METHOD M_AlarmManagement
//////////////////
// Manages Sepam Alarms. Alarms opens HT CB until Sepam manual Reset. Warning Opens CB-L but does not maintain warning.
/////////////////

VAR 
	// Method local variables (reinitialized at each cycle) 
	FB_AlarmCodeManager 	: FB_AlarmCodeManager; 
 	ComWarning				: BOOL;
	ComAlarms				: BOOL;
END_VAR
// ALARM CODE //
	FB_AlarmCodeManager(
		bAlarm1			:= MesDataExd.MesData.MesAlarmCom,			// Com alarm
		bAlarm2			:= MesDataExd.MesData.MesFault_Major,				// True := Major fault : cannot recover
		bAlarm3			:= MesDataExd.MesData.MesAlarm_AcOff,				// True := AC off		
		bAlarm4			:= MesDataExd.MesData.MesAlarm_GeneralOff,			// True := Imminent shut down
		bAlarm5			:= MesDataExd.MesData.MesFault_Bat,					// True := Battery disconnected
		bAlarm6			:= MesDataExd.MesData.MesFault_Charger,				// True := Charger out of order										 
		bAlarm7			:= MesDataExd.MesData.MesFault_12V,					// True := 12V absent 
		bAlarm8			:= MesDataExd.MesData.MesFault_48V,					// True := 48V absent
		bAlarm9			:= MesDataExd.MesData.MesToggleRead,				// True := AC power supply low 
		bAlarm10		:= FALSE, 									//										
		bAlarm11		:= FALSE,                                   //
		bAlarm12		:= FALSE,                                   //
		bAlarm13		:= FALSE,                                   //
		bAlarm14		:= FALSE,                                   //
		bAlarm15		:= FALSE, 									// 
		wAlarmCode		=>MesDataExd.MesData.MesAlarmCode);		

// WARNING CODE //
	FB_AlarmCodeManager(
		bAlarm1			:= MesDataExd.MesData.MesFault_Minor,				// True := Minor fault (overtemp, overcurrent, overvolt)
		bAlarm2			:= MesDataExd.MesData.MesAlarm_Ulow ,		// Battery  Capacity is low 
		bAlarm4			:= FALSE,									//
		bAlarm5			:= FALSE,									//
		bAlarm6			:= FALSE,									//
		bAlarm7			:= FALSE,									// 
		bAlarm8			:= FALSE,									// 
		bAlarm9			:= FALSE,									// 
		bAlarm10		:= FALSE,									// 
		bAlarm11		:= FALSE,									// 
		bAlarm12		:= FALSE,									// 
		bAlarm13		:= FALSE,									// 
		bAlarm14		:= FALSE,									// 
		bAlarm15		:= FALSE,									// 
		wAlarmCode		=>MesDataExd.MesData.MesWarningCode);					

// EVENT CODE //
	FB_AlarmCodeManager(
		bAlarm1			:=FALSE, 									// 
		bAlarm2			:=FALSE, 									// 
		bAlarm3			:=FALSE, 									// 
		bAlarm4			:=FALSE, 									// 
		bAlarm5			:=FALSE, 									//
		bAlarm6			:=FALSE,        							//
		bAlarm7			:=FALSE,        							//
		bAlarm8			:=FALSE,        							//
		bAlarm9			:=FALSE,        							//
		bAlarm10		:=FALSE, 									//
		bAlarm11		:=FALSE,        							//
		bAlarm12		:=FALSE,        							//
		bAlarm13		:=FALSE,        							//
		bAlarm14		:=FALSE,        							//
		bAlarm15		:=FALSE, 									//
		wAlarmCode		=> MesDataExd.MesData.MesEventCode);
END_METHOD

METHOD M_Evaluate
VAR_INPUT
END_VAR

VAR
END_VAR
END_METHOD

METHOD M_Read
//////////////////
//  Method Calls 
/////////////////

VAR_INPUT
	
END_VAR
VAR 
	MW					: FB_MergeWordsToFloat;
	MW_1				: FB_MergeWordsToDint;
END_VAR
// CP-Read / Write 


IF MesDataExd.MesData.MesCP_Read  THEN		
	
	FB_ModbusRead[1]
		(
			nTCPPort		:= ParamTcpPort,
			ClockRead		:= MesDataExd.MesData.MesCP_Read AND ClockRead, 
			Reset			:= CmdClearFault_G OR IN_CmdReset_L,
			sIPAddr			:= ParamIPAddress ,
			nUnitID			:= 1, 
			tTimeout		:= T#5S,
			nQuantity		:= 1, 
			nMBAddr			:= 44000 , 
			cbLength		:= SIZEOF(MesBlock1_Temp) , 
			pDestAddr		:= ADR(MesBlock1_Temp) , 
			ModbusReadAlarm	=> AX_ModbusReadAlarm[1] , 
			ErrorId			=> AX_ModbusReadAlarmId[1]
		);
		
	FB_ModbusRead[2]
		(
			nTCPPort		:= ParamTcpPort,
			ClockRead		:= MesDataExd.MesData.MesCP_Read AND ClockRead, 
			Reset			:= CmdClearFault_G OR IN_CmdReset_L,
			sIPAddr			:= ParamIPAddress ,
			nUnitID			:= 1, 
			tTimeout		:= T#5S,
			nQuantity		:= 9, 
			nMBAddr			:= 44100 , 
			cbLength		:= SIZEOF(MesBlock2_Temp) , 
			pDestAddr		:= ADR(MesBlock2_Temp) , 
			ModbusReadAlarm	=> AX_ModbusReadAlarm[2], 
			ErrorId			=> AX_ModbusReadAlarmId[2]
		);
		
	FB_ModbusRead[3]
		(
			nTCPPort		:= ParamTcpPort,
			ClockRead		:= MesDataExd.MesData.MesCP_Read AND ClockRead	, 
			Reset			:= CmdClearFault_G OR IN_CmdReset_L,
			sIPAddr			:= ParamIPAddress ,
			nUnitID			:= 1, 
			tTimeout		:= T#5S,
			nQuantity		:= 6, 
			nMBAddr			:= 44150 , 
			cbLength		:= SIZEOF(MesBlock3_Temp) , 
			pDestAddr		:= ADR(MesBlock3_Temp) , 
			ModbusReadAlarm	=> AX_ModbusReadAlarm[3], 
			ErrorId			=> AX_ModbusReadAlarmId[3]
		);
	
	FB_ModbusRead[4]
		(
			nTCPPort		:= ParamTcpPort,
			ClockRead		:= MesDataExd.MesData.MesCP_Read AND ClockRead, 
			Reset			:= CmdClearFault_G OR IN_CmdReset_L,
			sIPAddr			:= ParamIPAddress,
			nUnitID			:= 1, 
			tTimeout		:= T#5S,
			nQuantity		:= 2, 
			nMBAddr			:= 44050 , 
			cbLength		:= SIZEOF(MesBlock4_Temp) , 
			pDestAddr		:= ADR(MesBlock4_Temp) , 
			ModbusReadAlarm	=> AX_ModbusReadAlarm[4], 
			ErrorId			=> AX_ModbusReadAlarmId[4]
		);
		
	//COM
	MesDataExd.MesData.MesAlarmCom 			:= NOT WORD_TO_BOOL(MesBlock1_Temp[1]);
	MesDataExd.MesSoc						:= WORD_TO_REAL(MesBlock2_Temp[1])* 0.01;
	
	MW( WORD_STRONG:= MesBlock2_Temp[3  ],	WORD_WEAK := MesBlock2_Temp[2  ], VAR_OUT := MesDataExd.MesSoc);
	MW( WORD_STRONG:= MesBlock2_Temp[5  ],	WORD_WEAK := MesBlock2_Temp[4  ], VAR_OUT := MesDataExd.MesUdc_48V);
	MW( WORD_STRONG:= MesBlock2_Temp[7  ],	WORD_WEAK := MesBlock2_Temp[6  ], VAR_OUT := MesDataExd.MesUdc_12V);
	MW( WORD_STRONG:= MesBlock2_Temp[9  ],	WORD_WEAK := MesBlock2_Temp[8  ], VAR_OUT := MesDataExd.MesUBatt);
	MW( WORD_STRONG:= MesBlock2_Temp[11 ],	WORD_WEAK := MesBlock2_Temp[10 ], VAR_OUT := MesDataExd.MesIdc_Bat);

	MW( WORD_STRONG:= MesBlock3_Temp[2  ],	WORD_WEAK := MesBlock3_Temp[1  ], VAR_OUT := MesDataExd.MesDischarge);
	MesDataExd.MesEbackUp		  		:= WORD_TO_REAL(MesBlock3_Temp[3  ]) * 0.01;
	MesDataExd.MesEBackUpEna	  		:= WORD_TO_BOOL(MesBlock3_Temp[4  ]);
	MesDataExd.MesBatTestPer	  		:= WORD_TO_BOOL(MesBlock3_Temp[5  ]);
	MesDataExd.MesVacTripSelect	  		:= WORD_TO_BOOL(MesBlock3_Temp[6  ]);	
	MW( WORD_STRONG:= MesBlock3_Temp[8  ],	WORD_WEAK := MesBlock3_Temp[7  ], VAR_OUT := MesDataExd.MesCapacity_Nom);
	
	MesDataExd.MesFault_Minor 			:= MesBlock4_Temp[1].8;
	MesDataExd.MesFault_Major  		:= MesBlock4_Temp[1].11;
	MesDataExd.MesAlarm_AcOff 			:= MesBlock4_Temp[2].0;
	MesDataExd.MesAlarm_GeneralOff		:= MesBlock4_Temp[2].1;
	MesDataExd.MesData.MesAlarm_Ulow	:= MesBlock4_Temp[2].2;
	MesDataExd.MesFault_Bat			:= MesBlock4_Temp[2].3;
//		MesDataExd.MesFault_Bat			:= MesBlock4_Temp[2].4;
	MesDataExd.MesFault_12V			:= MesBlock4_Temp[2].5;
	MesDataExd.MesFault_48V			:= MesBlock4_Temp[2].6;
	MesDataExd.MesAlarm_AcLow			:= MesBlock4_Temp[2].7; 
		
END_IF 

	// properties update 
MesDataExd.MesData.MesUdc 				:= MesDataExd.MesUdc_12V ; 
MesDataExd.MesData.MesDischarging 		:= MesDataExd.MesAlarm_AcOff 	; 
	
MesDataExd.MesData.MesAlarmState 		:= MesDataExd.MesFault_Minor OR MesDataExd.MesFault_Major OR MesDataExd.MesAlarm_GeneralOff OR 
											 MesDataExd.MesFault_Bat OR MesDataExd.MesFault_Bat  ;
END_METHOD

END_FUNCTION_BLOCK

// ---- 01_Equipement_Library/UPS/FB_UPS_CXC.TcPOU
FUNCTION_BLOCK FB_UPS_CXC EXTENDS FB_UPS_Base
//////////////////
// UPS 
//////////////////
VAR_INPUT PERSISTENT
	// Parameters of the Object (instance/model specific) 

		{attribute 'OPC.UA.DA' := '1'} 
		ParamIPAddress				: STRING 	:= '192.168.20.66'; 	// (NA)Config: IP Adress of PV INverter
		{attribute 'OPC.UA.DA' := '1'} 
		ParamUnitID 				: BYTE  	:= 1; 			  		// (NA)   Modbus Unit ID. 
		{attribute 'OPC.UA.DA' := '1'} 
		ParamTCPPort				: UINT		:= 502;					// (NA) TCP port for modbus
		
END_VAR

VAR_OUTPUT
	//Child objects
	
END_VAR

VAR_INPUT
	// I/O Inputs
		IN_MesCbUPS_IO					: BOOL ; // 1 = opened. 
		
				MesDataExd						AT %Q*	: UPS_CXC ; 
		
END_VAR

VAR
	//M_ALARMMANAGEMENT VARIABLES//

	//M_READ//

		AX_ModbusRead		   		: ARRAY [1..2] OF FB_ModbusRead ; 					// (NA) FB for Modbus Reading
		ModbusReadInput				: FB_ModbusReadInput ; 		       
                                 
		MesBlock_Temp 				: ARRAY [1..2] OF ARRAY[1..120]  OF WORD; 			// (NA) Temporary Block with multiple modbus reading (Caution : Double Word variables)
		MesBlockInput				: ARRAY[1..1] OF BYTE ; 
		
	
	//M_EXECUTE //

		
END_VAR

METHOD M_AlarmManagement
//////////////////
// Manages Sepam Alarms. Alarms opens HT CB until Sepam manual Reset . Warning Opens CB-L but does not maintain warning
/////////////////

VAR 
	// Method local variables (reinitialized at each cycle) 
	FB_AlarmCodeManager 	: FB_AlarmCodeManager ; 

 
END_VAR
	//Alarm
	
	TON_ComAlarm	(IN:= (AX_ModbusRead[1].ModbusReadAlarm) AND (AX_ModbusRead[2].ModbusReadAlarm) AND (ModbusReadInput.ModbusReadAlarm) , PT:= ParamTempoComAlarm, 	Q=>MesDataExd.MesData.MesAlarmCom) ;	
	TON_ComWarning	(IN:= (AX_ModbusRead[1].ModbusReadAlarm) OR  (AX_ModbusRead[2].ModbusReadAlarm) OR  (ModbusReadInput.ModbusReadAlarm) , PT:= ParamTempoComWarning, 	Q=>MesWarningCom) ;	


// ALARM CODE //
	FB_AlarmCodeManager(
		bAlarm1				:= FALSE , 				 									//  
		bAlarm2				:= MesDataExd.MesData.MesAlarm_Ulow ,						// Battery SoC is low
		bAlarm3				:= MesDataExd.MesData.MesAlarmState ,					// UPS Fault synthesis
		bAlarm4				:= MesDataExd.MesOverTempBatt,     							// Battery overtemperature
		bAlarm5				:= FALSE,         											// 
		bAlarm6				:= FALSE, 													//
		bAlarm7				:= FALSE, 													//
		bAlarm8				:= FALSE,                                                   //
		bAlarm9				:= FALSE,                                                   //
		bAlarm10			:= FALSE,                                                   //
		bAlarm11			:= FALSE,                                                   //
		bAlarm12			:= FALSE,                                                   //
		bAlarm13			:= FALSE,                                                   //
		bAlarm14			:= FALSE,                                                   //
		bAlarm15			:= FALSE , 													//
		wAlarmCode			=> MesDataExd.MesData.MesAlarmCode);

// WARNING CODE //
	FB_AlarmCodeManager(
		bAlarm1			:= MesDataExd.MesData.MesDischarging , 				 			// UPS is discharging  , 														// 
		bAlarm2			:= MesDataExd.MesCBUpsOpened, 									// CB UPS Opened . 
		bAlarm3			:= MesWarningCom, 												// Communication warning  #COM
		bAlarm4			:= MesDataExd.MesData.MesAlarmCom,         						// Communication alarm, 	#COM													// 
		bAlarm5			:= FALSE, 														//
		bAlarm6			:= FALSE,                                                       //
		bAlarm7			:= FALSE,                                                       //
		bAlarm8			:= FALSE,                                                       //
		bAlarm9			:= FALSE,                                                       //
		bAlarm10		:= FALSE,                                                       //
		bAlarm11		:= FALSE,                                                       //
		bAlarm12		:= FALSE,                                                       //
		bAlarm13		:= FALSE,                                                       //
		bAlarm14		:= FALSE,                                                       //
		bAlarm15		:= FALSE,                                                       //
		wAlarmCode		=> MesDataExd.MesData.MesWarningCode);

// EVENT CODE //
	FB_AlarmCodeManager(
		bAlarm1			:=FALSE, 													// 
		bAlarm2			:=FALSE, 													// 
		bAlarm3			:=FALSE, 													// 
		bAlarm4			:=FALSE, 													// 
		bAlarm5			:=FALSE, 													//
		bAlarm6			:=FALSE,        											//
		bAlarm7			:=FALSE,        											//
		bAlarm8			:=FALSE,        											//
		bAlarm9			:=FALSE,        											//
		bAlarm10		:=FALSE,        											//
		bAlarm11		:=FALSE,        											//
		bAlarm12		:=FALSE,        											//
		bAlarm13		:=FALSE,        											//
		bAlarm14		:=FALSE,        											//
		bAlarm15		:=FALSE,        											//
		wAlarmCode		=> MesDataExd.MesData.MesEventCode);
END_METHOD

METHOD M_Read
//////////////////
//  Read Modbus Variable for PCS . 
/////////////////
VAR 
	// Method local variables (reinitialized at each cycle) 
		
		AX_Addr				: ARRAY[1..3] OF UINT := [16#82, 		16#C2, 	16#101];
		AX_Qty				: ARRAY[1..3] OF UINT := [16, 		6, 	4];
		
		MW 					: FB_MergeWordsToDint; 
END_VAR
// CP-Read / Write 


IF MesDataExd.MesData.MesCP_Read  THEN	

AX_ModbusRead[1]
(
	pDestAddr 		:= ADR(MesBlock_Temp[1]),
	sIPAddr 		:= ParamIPAddress,
	tTimeout 		:= ParamTimeout,
	nQuantity 		:= AX_Qty[1],
	ntcpport 		:= ParamTCPPort,
	nMBAddr 		:= AX_Addr[1]-2,
	nUnitID 		:= ParamUnitID,
	cbLength 		:= SIZEOF(MesBlock_Temp[1]),
	ClockRead 		:= ClockRead AND MesDataExd.MesData.MesCP_Read,
	Reset 			:= CmdClearFault_G OR IN_CmdReset_L,
);


AX_ModbusRead[2]
(
	pDestAddr 		:= ADR(MesBlock_Temp[2]),
	sIPAddr 		:= ParamIPAddress,
	tTimeout 		:= ParamTimeout,
	nQuantity 		:= AX_Qty[2],
	ntcpport 		:= ParamTCPPort,
	nMBAddr 		:= AX_Addr[2]-2,
	nUnitID 		:= ParamUnitID,
	cbLength 		:= SIZEOF(MesBlock_Temp[2]),
	ClockRead 		:= ClockRead AND MesDataExd.MesData.MesCP_Read,
	Reset 			:= CmdClearFault_G OR IN_CmdReset_L
);


ModbusReadInput
(
	pDestAddr 		:= ADR(MesBlockInput),
	sIPAddr 		:= ParamIPAddress,
	tTimeout 		:= ParamTimeout,
	nQuantity 		:= AX_Qty[3],
	ntcpport 		:= ParamTCPPort,
	nMBAddr 		:= AX_Addr[3]-1,
	nUnitID 		:= ParamUnitID,
	cbLength 		:= SIZEOF(MesBlockInput),
	ClockRead 		:= ClockRead AND MesDataExd.MesData.MesCP_Read,
	Reset 			:= GVL_CFG.CmdClearFault_G OR IN_CmdReset_L
);


	


MW(WORD_STRONG:= MesBlock_Temp[1][3], WORD_WEAK := MesBlock_Temp[1][4],SIGNED:=TRUE, FIX:=2 , SIZE:=2, VAR_OUT:=MesDataExd.MesIload);
MW(WORD_STRONG:= MesBlock_Temp[1][5], WORD_WEAK := MesBlock_Temp[1][6],SIGNED:=TRUE, FIX:=2 , SIZE:=2, VAR_OUT:=MesDataExd.MesUBatt);
MW(WORD_STRONG:= MesBlock_Temp[1][7], WORD_WEAK := MesBlock_Temp[1][8],SIGNED:=TRUE, FIX:=2 , SIZE:=2, VAR_OUT:=MesDataExd.MesIBatt);
MW(WORD_STRONG:= MesBlock_Temp[1][15], WORD_WEAK := MesBlock_Temp[1][16],SIGNED:=TRUE, FIX:=2 , SIZE:=2, VAR_OUT:=MesDataExd.MesSoC);

MW(WORD_STRONG:= MesBlock_Temp[2][1], WORD_WEAK := MesBlock_Temp[2][2],SIGNED:=TRUE, FIX:=2 , SIZE:=2, VAR_OUT:=MesDataExd.MesIdc);
MW(WORD_STRONG:= MesBlock_Temp[2][3], WORD_WEAK := MesBlock_Temp[2][4],SIGNED:=TRUE, FIX:=2 , SIZE:=2, VAR_OUT:=MesDataExd.MesData.MesUdc);
MW(WORD_STRONG:= MesBlock_Temp[2][5], WORD_WEAK := MesBlock_Temp[2][6],SIGNED:=TRUE, FIX:=2 , SIZE:=2, VAR_OUT:=MesDataExd.MesU);

MesDataExd.MesData.MesAlarm_Ulow := MesBlockInput[1].1	; // Low battery capacity 
MesDataExd.MesOverTempBatt	:= MesBlockInput[1].2 ; // OverTemp battery 
MesDataExd.MesData.MesDischarging := MesBlockInput[1].3 OR IN_MesDischarging_IO ; 
MesDataExd.MesData.MesAlarmState := IN_MesFault_IO ; 


END_IF


IF ParamNC THEN
	MesDataExd.MesCBUpsOpened := IN_MesCbUPS_IO ; 
	
ELSE 
 	MesDataExd.MesCBUpsOpened := NOT IN_MesCbUPS_IO ;
END_IF
END_METHOD

END_FUNCTION_BLOCK

// ---- 01_Equipement_Library/UPS/FB_UPS_Eneris.TcPOU
FUNCTION_BLOCK FB_UPS_ENERIS EXTENDS FB_UPS_Base
//////////////////
// UPS 
//////////////////
VAR_INPUT PERSISTENT
	// Parameters of the Object (instance/model specific) 
	ParamNC_Discharging					: BOOL := FALSE; 	(* (NA)False: TRUE = Closed, True : TRUE = opened*)
	ParamNC_Alarm_Ulow					: BOOL := FALSE; 	(* (NA)False: TRUE = Closed, True : TRUE = opened*)
	ParamNC_AlarmState					: BOOL := FALSE; 	(* (NA)False: TRUE = Closed, True : TRUE = opened*)
END_VAR

VAR_OUTPUT
	//Child objects
	
END_VAR

VAR_INPUT
	// I/O Inputs
		IN_MesCbUPS_IO					: BOOL ; // 1 = opened. 
		
			MesDataExd				: UPS_ENERIS ; 
	
		
END_VAR

VAR
	//M_ALARMMANAGEMENT VARIABLES//
		
	//M_READ//


		
	//M_EXECUTE //
		
	
END_VAR

METHOD M_AlarmManagement
//////////////////
// Manages Sepam Alarms. Alarms opens HT CB until Sepam manual Reset . Warning Opens CB-L but does not maintain warning
/////////////////

VAR 
	// Method local variables (reinitialized at each cycle) 
	FB_AlarmCodeManager 	: FB_AlarmCodeManager ; 

 
END_VAR
IF ParamNC_Discharging THEN 
	MesDataExd.MesData.MesDischarging  	:=  NOT IN_MesDischarging_IO;
ELSE
	MesDataExd.MesData.MesDischarging  	:=  IN_MesDischarging_IO;
END_IF

IF ParamNC_Alarm_Ulow THEN 
	MesDataExd.MesData.MesAlarm_Ulow 	 	:=  NOT IN_MesBatLow_IO;
ELSE
	MesDataExd.MesData.MesAlarm_Ulow 	 	:=  IN_MesBatLow_IO;
END_IF

IF ParamNC_AlarmState THEN 
	MesDataExd.MesData.MesAlarmState 		:=  NOT IN_MesFault_IO;
ELSE
	MesDataExd.MesData.MesAlarmState 		:=  IN_MesFault_IO;
END_IF

// ALARM CODE //
	FB_AlarmCodeManager(
		bAlarm1				:= FALSE , 				 						// 
		bAlarm2				:= MesDataExd.MesData.MesAlarm_Ulow ,						// Battery SoC is low 
		bAlarm3				:= MesDataExd.MesData.MesAlarmState ,						// UPS Fault synthesis		
		bAlarm4				:= FALSE,     									// 
		bAlarm5				:= FALSE,         								//  
		bAlarm6				:= FALSE, 										// 
		bAlarm7				:= FALSE,                                       //
		bAlarm8				:= FALSE,                                       //
		bAlarm9				:= FALSE,                                       //
		bAlarm10			:= FALSE,                                       //
		bAlarm11			:= FALSE,                                       //
		bAlarm12			:= FALSE,                                       //
		bAlarm13			:= FALSE,                                       //
		bAlarm14			:= FALSE,                                       //
		bAlarm15			:= FALSE ,	 									//
		wAlarmCode			=>MesDataExd.MesData.MesAlarmCode);

// WARNING CODE //
	FB_AlarmCodeManager(
		bAlarm1			:= MesDataExd.MesData.MesDischarging , 				 		// UPS is discharging  		
		bAlarm2			:= FALSE, 											// 
		bAlarm3			:= FALSE, 											// 
		bAlarm4			:= FALSE, 											// 
		bAlarm5			:= FALSE, 											//
		bAlarm6			:= FALSE,                                           //
		bAlarm7			:= FALSE,                                           //
		bAlarm8			:= FALSE,                                           //
		bAlarm9			:= FALSE,                                           //
		bAlarm10		:= FALSE,                                           //
		bAlarm11		:= FALSE,                                           //
		bAlarm12		:= FALSE,                                           //
		bAlarm13		:= FALSE,                                           //
		bAlarm14		:= FALSE,                                           //
		bAlarm15		:= FALSE,                                           //
		wAlarmCode		=>MesDataExd.MesData.MesWarningCode);

// EVENT CODE //
	FB_AlarmCodeManager(
		bAlarm1			:=FALSE, 											// 
		bAlarm2			:=FALSE, 											// 
		bAlarm3			:=FALSE, 											// 
		bAlarm4			:=FALSE, 											// 
		bAlarm5			:=FALSE, 											//
		bAlarm6			:=FALSE, 											//
		bAlarm7			:=FALSE, 											//
		bAlarm8			:=FALSE, 											//
		bAlarm9			:=FALSE, 											//
		bAlarm10		:=FALSE, 											//
		bAlarm11		:=FALSE, 											//
		bAlarm12		:=FALSE, 											//
		bAlarm13		:=FALSE, 											//
		bAlarm14		:=FALSE, 											//
		bAlarm15		:=FALSE, 											//
		wAlarmCode		=>MesDataExd.MesData.MesEventCode);
END_METHOD

END_FUNCTION_BLOCK

// ---- 04_Application/Checks/CheckBounds.TcPOU
// Implicitly generated code : DO NOT EDIT
FUNCTION CheckBounds : DINT
VAR_INPUT
	index, lower, upper: DINT;
END_VAR

// Implicitly generated code : Only an Implementation suggestion
{noflow}

Fault_Count_G(CU:=FALSE) ; 
IF  index < lower THEN
	CheckBounds := lower;
	Fault_Count_G(CU:=TRUE) ; 
ELSIF  index > upper THEN
	CheckBounds := upper;
	Fault_Count_G(CU:=TRUE) ; 
ELSE  
	CheckBounds := index;
END_IF
{flow}

END_FUNCTION

// ---- 04_Application/Checks/CheckDivDInt.TcPOU
// Implicitly generated code : DO NOT EDIT
FUNCTION CheckDivDInt : DINT
VAR_INPUT
	divisor:DINT;
END_VAR

// Implicitly generated code : Only an Implementation suggestion
{noflow}
Fault_Count_G(CU:=FALSE) ; 
IF divisor = 0 THEN
	CheckDivDInt:=1;
		Fault_Count_G(CU:=TRUE) ; 
ELSE
	CheckDivDInt:=divisor;
END_IF;
{flow}

END_FUNCTION

// ---- 04_Application/Checks/CheckDivLInt.TcPOU
// Implicitly generated code : DO NOT EDIT
FUNCTION CheckDivLInt : LINT
VAR_INPUT
	divisor:LINT;
END_VAR

// Implicitly generated code : Only an Implementation suggestion
{noflow}
Fault_Count_G(CU:=FALSE) ; 
IF divisor = 0 THEN
	CheckDivLInt:=1;
		Fault_Count_G(CU:=TRUE) ; 
ELSE
	CheckDivLInt:=divisor;
END_IF;
{flow}

END_FUNCTION

// ---- 04_Application/Checks/CheckDivLReal.TcPOU
// Implicitly generated code : DO NOT EDIT
FUNCTION CheckDivLReal : LREAL
VAR_INPUT
	divisor:LREAL;
END_VAR

// Implicitly generated code : Only an Implementation suggestion
{noflow}
Fault_Count_G(CU:=FALSE) ; 
IF divisor = 0 THEN
	CheckDivLReal:=1;
		Fault_Count_G(CU:=TRUE) ; 
ELSE
	CheckDivLReal:=divisor;
END_IF;
{flow}

END_FUNCTION

// ---- 04_Application/Checks/CheckDivReal.TcPOU
// Implicitly generated code : DO NOT EDIT
FUNCTION CheckDivReal : REAL
VAR_INPUT
	divisor:REAL;
END_VAR

// Implicitly generated code : Only an Implementation suggestion
{noflow}
Fault_Count_G(CU:=FALSE) ; 
IF divisor = 0 THEN
	CheckDivReal:=1;
		Fault_Count_G(CU:=TRUE) ; 
ELSE
	CheckDivReal:=divisor;
END_IF;
{flow}

END_FUNCTION

// ---- 04_Application/Checks/CheckLRangeSigned.TcPOU
// Implicitly generated code : DO NOT EDIT
FUNCTION CheckLRangeSigned : LINT
VAR_INPUT
	value, lower, upper: LINT;
END_VAR

// Implicitly generated code : Only an Implementation suggestion
{noflow}
Fault_Count_G(CU:=FALSE) ; 
IF (value < lower) THEN
	CheckLRangeSigned := lower;
		Fault_Count_G(CU:=TRUE) ; 
ELSIF(value > upper) THEN
	CheckLRangeSigned := upper;
		Fault_Count_G(CU:=TRUE) ; 
ELSE
	CheckLRangeSigned := value;
END_IF

{flow}

END_FUNCTION

// ---- 04_Application/Checks/CheckLRangeUnsigned.TcPOU
// Implicitly generated code : DO NOT EDIT
FUNCTION CheckLRangeUnsigned : ULINT
VAR_INPUT
	value, lower, upper: ULINT;
END_VAR

// Implicitly generated code : Only an Implementation suggestion
{noflow}
Fault_Count_G(CU:=FALSE) ; 
IF (value < lower) THEN
	CheckLRangeUnsigned := lower;
		Fault_Count_G(CU:=TRUE) ; 
ELSIF(value > upper) THEN
	CheckLRangeUnsigned := upper;
		Fault_Count_G(CU:=TRUE) ; 
ELSE
	CheckLRangeUnsigned := value;
END_IF
{flow}

END_FUNCTION

// ---- 04_Application/Checks/CheckPointer.TcPOU
// Code généré automatiquement : NE PAS MODIFIER
FUNCTION CheckPointer : POINTER TO BYTE
VAR_INPUT 
	ptToTest : POINTER TO BYTE; // Adresse de destination du pointeur
	iSize : DINT;		        // Taille du type indiqué par le pointeur.  (par exemple : 20 pour POINTER TO ARRAY [0..9] OF INT)
	iGran : DINT;		        // Granularité de l’accès au pointeur. Il s’agit de la taille du plus grand type de données non structuré dans le type indiqué par le pointeur.  (par exemple : 2 pour POINTER TO ARRAY [0..9] OF INT)
	bWrite: BOOL;		        // Indique l’accès en lecture ou en écriture. TRUE = accès en écriture.
END_VAR

// Pas d’implémentation standard. Veuillez insérer votre code ici.
CheckPointer := ptToTest;
{flow}

END_FUNCTION

// ---- 04_Application/Checks/CheckRangeSigned.TcPOU
// Implicitly generated code : DO NOT EDIT
FUNCTION CheckRangeSigned : DINT
VAR_INPUT
	value, lower, upper: DINT;
END_VAR

// Implicitly generated code : Only an Implementation suggestion
{noflow}
Fault_Count_G(CU:=FALSE) ; 
IF (value < lower) THEN
	CheckRangeSigned := lower;
		Fault_Count_G(CU:=TRUE) ; 
ELSIF(value > upper) THEN
	CheckRangeSigned := upper;
		Fault_Count_G(CU:=TRUE) ; 
ELSE
	CheckRangeSigned := value;
END_IF
{flow}

END_FUNCTION

// ---- 04_Application/Checks/CheckRangeUnsigned.TcPOU
// Implicitly generated code : DO NOT EDIT
FUNCTION CheckRangeUnsigned : UDINT
VAR_INPUT
	value, lower, upper: UDINT;
END_VAR

// Implicitly generated code : Only an Implementation suggestion
{noflow}
Fault_Count_G(CU:=FALSE) ; 
IF (value < lower) THEN
	CheckRangeUnsigned := lower;
		Fault_Count_G(CU:=TRUE) ; 
ELSIF(value > upper) THEN
	CheckRangeUnsigned := upper;
		Fault_Count_G(CU:=TRUE) ; 
ELSE
	CheckRangeUnsigned := value;
END_IF
{flow}

END_FUNCTION

// ---- 04_Application/EMS/PRG_EMS.TcPOU
PROGRAM PRG_EMS
VAR_INPUT
	IN_CmdRebootEMS							: BOOL;
	IN_CmdKillEMS							: BOOL;
	MesData									: EMS;
END_VAR
VAR_INPUT PERSISTENT
	
	ParamTimeKeepReboot						: TIME := T#1M;
	ParamTimeKeepSetptFromGrid				: TIME := T#15M;
	ParamTimeout_Warning					: TIME := T#10M;
	ParamTimeout_Alarm						: TIME := T#1H;
	
END_VAR


VAR PERSISTENT
	
	DT_Time_EMS_ApplyNextSetpoint			: DT;
	SetptP_Grid 							: REAL;
	SetptP_Grid_Min							: REAL;
	SetptP_Grid_Max  						: REAL;
	IN_EMS 									: IN_EMS;		// Structure sent by EMS
	
END_VAR

VAR
	
	OUT_EMS 								: OUT_EMS;		// Structure sent to the EMS
	                    					
	AX_SystemBms_1_1 						: BAT;
	AX_SystemBms_1_2 						: BAT;
	                    					
	KK										: INT;
	Watchdog_Old							: REAL;
	RS_Penalties							: RS;
	                    					
	IN_EMS_OLD								: IN_EMS;
	                    	
	Average_PGrid							: FB_Average;
	Average_Pbat							: FB_Average;
	Average_Psol							: FB_Average;
	InitialCalc								: BOOL;
	
	TRIG_NewSetptFromGrid					: R_TRIG;
	TON_MaintainSetptGrid					: TON;
	F_TRIG_TON_MaintainSetptGrid			: F_TRIG;
	RS_MaintainRequest						: RS;
	                                    	
	TP_Reboot								: TP;
	TP_KillEms								: TP;
	TON_TimeoutAlarm						: TON;
	TON_TimeoutWarning						: TON;
	
	TRIG_ApplySetpoint						: R_TRIG;
	
	DT_Time_Now								: DT;
	
	
	TIME_ApplySetpoint						: TIMESTRUCT;
	

	
	xTestTime								: DATE_AND_TIME;
	xTestTime1								: DATE_AND_TIME;
	xTestTime2								: DATE_AND_TIME;
	xTestReal								: REAL;
END_VAR



M_Evaluate();
M_AlarmManagement();

METHOD M_AlarmManagement : BOOL
VAR
	FB_AlarmCodeManager : FB_AlarmCodeManager;
END_VAR
	
// ALARM CODE //
	FB_AlarmCodeManager(
		bAlarm1				:= TP_Reboot.Q, 			// Reboot order
		bAlarm2				:= TP_KillEms.Q,			// Kill EMS order
		bAlarm3				:= TON_TimeoutWarning.Q , 	// No EMS update Warning : Timeout for EMS
		bAlarm4				:= TON_TimeoutAlarm.Q , 	// No EMS update Alarm : Critical timeout for EMS
		bAlarm5				:= FALSE, 					//			 
		bAlarm6				:= FALSE, 					//			 
		bAlarm7				:= FALSE,       			//
		bAlarm8				:= FALSE,       			//
		bAlarm9				:= FALSE,       			//
		bAlarm10			:= FALSE,       			//
		bAlarm11			:= FALSE, 					//			
		bAlarm12			:= FALSE,       			//
		bAlarm13			:= FALSE,       			//
		bAlarm14			:= FALSE, 					//	
		bAlarm15			:= FALSE ,   				// 
		wAlarmCode			=> MesData.MesAlarmCode);
END_METHOD

METHOD M_Evaluate : BOOL
VAR_INPUT
END_VAR

VAR
	LL: INT;
	KK : INT;
	EE : INT;
	PP : INT;
END_VAR
// Gestion des Inputs venant de l'EMS
	MesData.IN_EMS := IN_EMS;

	TP_Reboot(IN := IN_CmdRebootEMS, pt := ParamTimeKeepReboot);
	TP_KillEms(IN := IN_CmdKillEMS, PT := ParamTimeKeepReboot);
	
	IF IN_CmdRebootEMS THEN
		IN_CmdRebootEMS := FALSE;
	END_IF
	IF IN_CmdKillEMS THEN
		IN_CmdKillEMS := FALSE;
	END_IF
	

	
	RS_Penalties(SET := A1_SUBMV.A1_ProtectRelay.MesDataExd.MesData.MesAlarmUmin, RESET1 := CalLocalTimeStruct.wHour = 0);
	
//	IF CalLocalTimeStruct.wMilliseconds < 30 AND CalLocalTimeStruct.wSecond = 0 AND CalLocalTimeStruct.wMinute MOD 10 = 0 THEN
		InitialCalc := TRUE;
		OUT_EMS.OUT_MesP_GRID := Average_PGrid.ValueOut;
		OUT_EMS.OUT_MesP_ESS := Average_Pbat.ValueOut;
		OUT_EMS.OUT_MesP_SPP := Average_Psol.ValueOut;
//	END_IF

	
	IF InitialCalc THEN
		Average_PGrid(ValueIn := A1_PP.MesData.MesPgrid, WindowDuration := 600000);
		Average_Pbat(ValueIn := A1_PP.MesData.MesPbat, WindowDuration := 600000);
		Average_Psol(ValueIn := A1_PP.MesData.MesPsol, WindowDuration := 600000);
	END_IF

	
// Gestion des Outputs à envoyer à l'EMS

	IF Watchdog_Old <> IN_EMS.IN_Watchdog THEN
		Watchdog_Old := IN_EMS.IN_Watchdog;
		OUT_EMS.OUT_Watchdog := IN_EMS.IN_Watchdog+1;
	END_IF
	OUT_EMS.OUT_MesAvailability_SPP	 := A1_PP.MesData.MesPsol_Connected/A1_PP.ParamPsolmax;

	
	OUT_EMS.OUT_CmdRebootEMS						:= TP_Reboot.Q;
	
	
	OUT_EMS.OUT_SetptP_GRID							:= A1_SUBMV.A1_GRID.MesDataExd.MesData.OUT_SetptP;
	OUT_EMS.OUT_NoPenalties							:= RS_Penalties.Q1;
	
	MesData.OUT_EMS := OUT_EMS;

// Alarm & Warning de perte de communication entre IPC SCADA et IPC EMS  

	TON_TimeoutAlarm(in := MEMCMP(pBuf1 := ADR(IN_EMS), pBuf2 := ADR(IN_EMS_OLD), n:=SIZEOF(IN_EMS)) = 0, PT := ParamTimeout_Alarm);
	TON_TimeoutWarning(in := MEMCMP(pBuf1 := ADR(IN_EMS), pBuf2 := ADR(IN_EMS_OLD), n:=SIZEOF(IN_EMS)) = 0, PT := ParamTimeout_Warning);
	
	IF MEMCMP(pBuf1 := ADR(IN_EMS), pBuf2 := ADR(IN_EMS_OLD), n:=SIZEOF(IN_EMS))<>0 THEN
		MEMCPY(srcAddr := ADR(IN_EMS), destAddr := ADR(IN_EMS_OLD), n:= SIZEOF(in_ems));
	END_IF
	
		A1_PP.IN_SetptP_GRID_min	:= SetptP_Grid_Min;
		A1_PP.IN_SetptP_GRID_max	:= SetptP_Grid_Max;
		//A1_PP.IN_SetptP_GRID_max:=xTestReal;
		//IN_EMS.IN_SetptP_GRID_max:=xTestReal;
		
	A1_PP.IN_SetptP_SPP_Remote := MAX(A1_PP.IN_SetptP_GRID_max + ABS(A1_PP.MesData.MesPbatCharge_Connected), 0);
	IF SetptP_Grid <= A1_PP.MesData.MesPsol THEN //if the EMS septpt is less that solar availability thenthe PP setpoint will be the  one EMS sends, this way we can charge the batteries with the leftover solar energy
		A1_PP.IN_SetptP_PP_Remote := SetptP_Grid;
	ELSIF SetptP_Grid_Min <= A1_PP.MesData.MesPsol THEN //if the EMS setpt min is less than solar availability then we continue producing solar energy in order not to get too many penalities
		A1_PP.IN_SetptP_PP_Remote := A1_PP.MesData.MesPsol;
	ELSE
		A1_PP.IN_SetptP_PP_Remote := SetptP_Grid_Min;
	END_IF
	

//SOC Calibration

// Ajout de la Sécurité de l'EMS:
	IF A1_SUBMV.A1_GRID.MesDataExd.MesData.OUT_SetptP < 0.95 * A1_PP.ParamPmax THEN
		A1_PP.IN_SetptP_PP_Remote := MIN(A1_SUBMV.A1_GRID.MesDataExd.MesData.OUT_SetptP,SetptP_Grid);
	END_IF
	
	DT_Time_EMS_ApplyNextSetpoint := DINT_TO_DT(LINT_TO_DINT(IN_EMS.IN_TimeApplySetpoint_LINT));
	DT_Time_Now	:= systemtime_to_dt(TIMESTR := CalGMTTimeStruct);
	TRIG_ApplySetpoint(CLK := DT_Time_EMS_ApplyNextSetpoint <= DINT_TO_DT(DT_TO_DINT(DT_Time_Now) - A1_SUBMV.A1_GRID.MesDataExd.MesEcart_HeureGrid));
	
	IF TRIG_ApplySetpoint.Q THEN
		TIME_ApplySetpoint := CalLocalTimeStruct;
		SetptP_Grid := IN_EMS.IN_SetptP_GRID;
		SetptP_Grid_Min := IN_EMS.IN_SetptP_GRID_min;
		SetptP_Grid_Max := IN_EMS.IN_SetptP_GRID_max;
	END_IF
	
// Detection Ecretage

	OUT_EMS.OUT_Ecretage:=0;	
	
	IF A1_PP.MesData.OUT_SetptP_SPP_PID > A1_PP.MesData.MesPsol - ParamDeadBandEcretage AND A1_PP.MesData.OUT_SetptP_SPP_PID < A1_PP.MesData.MesPsol + ParamDeadBandEcretage THEN
		IF A1_PP.MesData.OUT_SetptP_SPP_PID < A1_PP.MesData.MesPsol_Connected - ParamDeadBandEcretage THEN 
			IF 0 <> A1_PP.MesData.MesPsol_Connected THEN
				OUT_EMS.OUT_Ecretage:=1;
			END_IF
		END_IF		
	END_IF
END_METHOD

END_PROGRAM

// ---- 04_Application/HMI/Infos/InfosIO.TcPOU
PROGRAM InfosIO
VAR_INPUT
END_VAR
VAR_OUTPUT
END_VAR
VAR

	
	bInit: BOOL := TRUE;
	KK: INT;
END_VAR

END_PROGRAM

// ---- 04_Application/HMI/Parameters/ParamBESS_HMI.TcPOU
PROGRAM ParamBESS_HMI
VAR
	
BESS_Num								: UINT;

// BESS
	BESS_TmpLowAlm						: REAL;	bOneBESS_TmpLowAlm						: BOOL;	bAllBESS_TmpLowAlm						: BOOL;
	BESS_TmpLowWarn						: REAL;	bOneBESS_TmpLowWarn						: BOOL;	bAllBESS_TmpLowWarn						: BOOL;
	BESS_TempHighAlm					: REAL;	bOneBESS_TempHighAlm					: BOOL;	bAllBESS_TempHighAlm					: BOOL;
	BESS_TempHighWarn					: REAL;	bOneBESS_TempHighWarn					: BOOL;	bAllBESS_TempHighWarn					: BOOL;
	BESS_HygroHighAlarm					: REAL;	bOneBESS_HygroHighAlarm					: BOOL;	bAllBESS_HygroHighAlarm					: BOOL;
	BESS_HygroHighWarn					: REAL;	bOneBESS_HygroHighWarn					: BOOL;	bAllBESS_HygroHighWarn					: BOOL;
	BESS_HygroStartHVAC					: REAL;	bOneBESS_HygroStartHVAC					: BOOL;	bAllBESS_HygroStartHVAC					: BOOL;
	BESS_HygroStopHvac					: REAL;	bOneBESS_HygroStopHvac					: BOOL;	bAllBESS_HygroStopHvac					: BOOL;
	BESS_TempStartHvac					: REAL;	bOneBESS_TempStartHvac					: BOOL;	bAllBESS_TempStartHvac					: BOOL;
	BESS_TempStopHvac					: REAL;	bOneBESS_TempStopHvac					: BOOL;	bAllBESS_TempStopHvac					: BOOL;
	BESS_Hvac_Setpt						: REAL;	bOneBESS_Hvac_Setpt						: BOOL;	bAllBESS_Hvac_Setpt						: BOOL;
	BESS_Hvac_TimeChangePrio			: TIME;	bOneBESS_Hvac_TimeChangePrio			: BOOL;	bAllBESS_Hvac_TimeChangePrio			: BOOL;
	BESS_TimeBatDoorOpened				: TIME;	bOneBESS_TimeBatDoorOpened				: BOOL;	bAllBESS_TimeBatDoorOpened				: BOOL;
	BESS_TimePcsDoorOpened				: TIME;	bOneBESS_TimePcsDoorOpened				: BOOL;	bAllBESS_TimePcsDoorOpened				: BOOL;

	


// SystemBMS
	SBMS1_ParamIpAddress				: STRING;
	SBMS1_ParamTcpPort					: UINT;
	SBMS1_ParamClockWriteTime			: TIME;
	SBMS2_ParamIpAddress				: STRING;
	SBMS2_ParamTcpPort					: UINT;
	SBMS2_ParamClockWriteTime			: TIME;

// HVAC
	HVAC1_ParamIpAddress				: STRING;
	HVAC1_ParamUnitId					: UINT;
	HVAC1_ParamTcpPort					: UINT;
	HVAC1_ParamClockWriteTime			: TIME;
	HVAC2_ParamIpAddress				: STRING;
	HVAC2_ParamUnitId					: UINT;
	HVAC2_ParamTcpPort					: UINT;
	HVAC2_ParamClockWriteTime			: TIME;	
	
// PCS
	PCS_RefreshValues						: BOOL;
	
	PCS1_ParamUnitID 						: BYTE  	;		PCS1_bParamUnitID 						: BOOL;	
	PCS1_ParamIPAddress			   			: STRING 	;       PCS1_bParamIPAddress			   		: BOOL;
	PCS1_ParamTcpPort						: UINT		;       PCS1_bParamTcpPort						: BOOL;
	PCS1_ParamNbPcs		            		: BYTE	 	;       PCS1_bParamNbPcs		            	: BOOL;
	PCS1_ParamTempoComAlarm					: TIME      ;       PCS1_bParamTempoComAlarm				: BOOL; 
	PCS1_ParamTempoComWarning				: TIME 		;       PCS1_bParamTempoComWarning				: BOOL;
	PCS1_ParamTimeOutBlckStrt          		: TIME 		;       PCS1_bParamTimeOutBlckStrt          	: BOOL;
	PCS1_ParamClockReadTime 				: TIME 		;       PCS1_bParamClockReadTime 				: BOOL;
	PCS1_ParamClockWriteTime 				: TIME      ;       PCS1_bParamClockWriteTime 				: BOOL;
	PCS1_ParamTimeout		            	: TIME 		;       PCS1_bParamTimeout		            	: BOOL;
	PCS1_ParamTimePulseTrig		    		: TIME 		;       PCS1_bParamTimePulseTrig		    	: BOOL;
	PCS1_ParamEssNum						: UINT      ;       PCS1_bParamEssNum						: BOOL;
	PCS1_ParamPcsNum						: UINT      ;		PCS1_bParamPcsNum						: BOOL;	
	PCS1_ParamPnom							: REAL      ;       PCS1_bParamPnom							: BOOL;
	PCS1_ParamQnom							: REAL 		;       PCS1_bParamQnom							: BOOL;
	PCS1_ParamTimeoutCmdQ					: TIME 		;       PCS1_bParamTimeoutCmdQ					: BOOL;
	PCS1_ParamTimeoutCmdCosPhi				: TIME		;       PCS1_bParamTimeoutCmdCosPhi				: BOOL;
	PCS1_ParamTimeoutQvU					: TIME      ;       PCS1_bParamTimeoutQvU					: BOOL;
	PCS1_ParamTimeoutPvF		        	: TIME      ;       PCS1_bParamTimeoutPvF		        	: BOOL;
	PCS1_ParamSetPtModbusMode				: BOOL      ;       PCS1_bParamSetPtModbusMode				: BOOL;
	PCS1_ParamPoverQ						: BOOL      ;       PCS1_bParamPoverQ						: BOOL;
	PCS1_ParamTimeSoCRangeReachedRmp		: TIME      ;       PCS1_bParamTimeSoCRangeReachedRmp		: BOOL;
	PCS1_ParamTimeFreqRegStbDuration		: TIME      ;       PCS1_bParamTimeFreqRegStbDuration		: BOOL;
	PCS1_ParamTimeEnterStblPriorRmp			: TIME      ;       PCS1_bParamTimeEnterStblPriorRmp		: BOOL;
	PCS1_ParamTimeoutGridFormerTransition	: TIME      ;       PCS1_bParamTimeoutGridFormerTransition	: BOOL;
	PCS1_ParamTimeoutGridFeederTransition	: TIME      ;       PCS1_bParamTimeoutGridFeederTransition	: BOOL;
	PCS1_ParamTimeoutOffTransition		    : TIME      ;       PCS1_bParamTimeoutOffTransition		    : BOOL;
	PCS1_ParamFreqRegSoCmax 				: REAL      ;       PCS1_bParamFreqRegSoCmax 				: BOOL;
	PCS1_ParamFreqRegSoCmin 			    : REAL      ;       PCS1_bParamFreqRegSoCmin 			    : BOOL;
	PCS1_ParamLVRT_Enabled					: BOOL      ;       PCS1_bParamLVRT_Enabled					: BOOL;
	PCS1_ParamAntiIslanding_Enabled			: BOOL      ;       PCS1_bParamAntiIslanding_Enabled		: BOOL;

	PCS2_ParamUnitID 						: BYTE  	;		PCS2_bParamUnitID 						: BOOL;		
	PCS2_ParamIPAddress			   			: STRING 	;       PCS2_bParamIPAddress			   		: BOOL;
	PCS2_ParamTcpPort						: UINT		;       PCS2_bParamTcpPort						: BOOL;
	PCS2_ParamNbPcs		            		: BYTE	 	;       PCS2_bParamNbPcs		            	: BOOL;
	PCS2_ParamTempoComAlarm					: TIME      ;       PCS2_bParamTempoComAlarm				: BOOL;      
	PCS2_ParamTempoComWarning				: TIME 		;       PCS2_bParamTempoComWarning				: BOOL;
	PCS2_ParamTimeOutBlckStrt          		: TIME 		;       PCS2_bParamTimeOutBlckStrt          	: BOOL;
	PCS2_ParamClockReadTime 				: TIME 		;       PCS2_bParamClockReadTime 				: BOOL;
	PCS2_ParamClockWriteTime 				: TIME      ;       PCS2_bParamClockWriteTime 				: BOOL;
	PCS2_ParamTimeout		            	: TIME 		;       PCS2_bParamTimeout		            	: BOOL;
	PCS2_ParamTimePulseTrig		    		: TIME 		;       PCS2_bParamTimePulseTrig		    	: BOOL;
	PCS2_ParamEssNum						: UINT      ;       PCS2_bParamEssNum						: BOOL;
	PCS2_ParamPcsNum						: UINT      ;		PCS2_bParamPcsNum						: BOOL;		
	PCS2_ParamPnom							: REAL      ;       PCS2_bParamPnom							: BOOL;
	PCS2_ParamQnom							: REAL 		;       PCS2_bParamQnom							: BOOL;
	PCS2_ParamTimeoutCmdQ					: TIME 		;       PCS2_bParamTimeoutCmdQ					: BOOL;
	PCS2_ParamTimeoutCmdCosPhi				: TIME		;       PCS2_bParamTimeoutCmdCosPhi				: BOOL;
	PCS2_ParamTimeoutQvU					: TIME      ;       PCS2_bParamTimeoutQvU					: BOOL;
	PCS2_ParamTimeoutPvF		        	: TIME      ;       PCS2_bParamTimeoutPvF		        	: BOOL;
	PCS2_ParamSetPtModbusMode				: BOOL      ;       PCS2_bParamSetPtModbusMode				: BOOL;
	PCS2_ParamPoverQ						: BOOL      ;       PCS2_bParamPoverQ						: BOOL;
	PCS2_ParamTimeSoCRangeReachedRmp		: TIME      ;       PCS2_bParamTimeSoCRangeReachedRmp		: BOOL;
	PCS2_ParamTimeFreqRegStbDuration		: TIME      ;       PCS2_bParamTimeFreqRegStbDuration		: BOOL;
	PCS2_ParamTimeEnterStblPriorRmp			: TIME      ;       PCS2_bParamTimeEnterStblPriorRmp		: BOOL;
	PCS2_ParamTimeoutGridFormerTransition	: TIME      ;       PCS2_bParamTimeoutGridFormerTransition	: BOOL;
	PCS2_ParamTimeoutGridFeederTransition	: TIME      ;       PCS2_bParamTimeoutGridFeederTransition	: BOOL;
	PCS2_ParamTimeoutOffTransition		    : TIME      ;       PCS2_bParamTimeoutOffTransition		    : BOOL;
	PCS2_ParamFreqRegSoCmax 				: REAL      ;       PCS2_bParamFreqRegSoCmax 				: BOOL;
	PCS2_ParamFreqRegSoCmin 			    : REAL      ;       PCS2_bParamFreqRegSoCmin 			    : BOOL;
	PCS2_ParamLVRT_Enabled					: BOOL      ;       PCS2_bParamLVRT_Enabled					: BOOL;
	PCS2_ParamAntiIslanding_Enabled			: BOOL      ;       PCS2_bParamAntiIslanding_Enabled		: BOOL;	
	
                                        
// QfU and PvF          
	bResetParamQfU_PvF					: BOOL;				// Reset Parameters                
	ParamQfU_UDbHigh    				: WORD;				// JEMA U1 : AKUO U_UDbHigh
	ParamQfU_Umax		    			: WORD;				// JEMA U2 : AKUO U_Umax
	ParamQfU_UDbLow	    				: WORD;				// JEMA U3 : AKUO U_UDbLow
	ParamQfU_Umin		    			: WORD;				// JEMA U4 : AKUO U_Umin
										
	ParamQfU_QDbHigh					: WORD;				// JEMA Q1 : AKUO U_QDbHigh
	ParamQfU_Qmax						: WORD;				// JEMA Q2 : AKUO U_Qmax
	ParamQfU_QDbLow						: WORD;				// JEMA Q3 : AKUO U_QDbLow
	ParamQfU_Qmin						: WORD;				// JEMA Q4 : AKUO U_Qmin
										
	ParamPfF_FDbHigh	    			: WORD;				// JEMA f1 : AKUO P_FDbHigh
	ParamPfF_Fmax		    			: WORD;				// JEMA f2 : AKUO P_Fmax
	ParamPfF_FDbLow	    				: WORD;				// JEMA f3 : AKUO P_FDbLow
	ParamPfF_Fmin		    			: WORD;				// JEMA f4 : AKUO P_Fmin
										
	ParamPfF_PDbHigh					: WORD;				// JEMA P1 : AKUO P_PDbHigh
	ParamPfF_Pmax						: WORD;				// JEMA P2 : AKUO P_Pmax
	ParamPfF_PDbLow						: WORD;				// JEMA P3 : AKUO P_PDbLow
	ParamPfF_Pmin						: WORD;				// JEMA P4 : AKUO P_Pmin

	ParamPfF_FhystLow					: WORD;				// JEMA fst1
	ParamPfF_FhystHigh					: WORD;				// JEMA fst2
	                                    

	ParamQfU_UDbHigh_HMI   				: REAL;				// JEMA U1 : AKUO U_UDbHigh
	ParamQfU_Umax_HMI	    			: REAL;				// JEMA U2 : AKUO U_Umax
	ParamQfU_UDbLow_HMI   				: REAL;				// JEMA U3 : AKUO U_UDbLow
	ParamQfU_Umin_HMI	    			: REAL;				// JEMA U4 : AKUO U_Umin
										
	ParamQfU_QDbHigh_HMI				: REAL;				// JEMA Q1 : AKUO U_QDbHigh
	ParamQfU_Qmax_HMI					: REAL;				// JEMA Q2 : AKUO U_Qmax
	ParamQfU_QDbLow_HMI					: REAL;				// JEMA Q3 : AKUO U_QDbLow
	ParamQfU_Qmin_HMI					: REAL;				// JEMA Q4 : AKUO U_Qmin
										
	ParamPfF_FDbHigh_HMI    			: REAL;				// JEMA f1 : AKUO P_FDbHigh
	ParamPfF_Fmax_HMI	    			: REAL;				// JEMA f2 : AKUO P_Fmax
	ParamPfF_FDbLow_HMI   				: REAL;				// JEMA f3 : AKUO P_FDbLow
	ParamPfF_Fmin_HMI	    			: REAL;				// JEMA f4 : AKUO P_Fmin
										
	ParamPfF_PDbHigh_HMI				: REAL;				// JEMA P1 : AKUO P_PDbHigh
	ParamPfF_Pmax_HMI					: REAL;				// JEMA P2 : AKUO P_Pmax
	ParamPfF_PDbLow_HMI					: REAL;				// JEMA P3 : AKUO P_PDbLow
	ParamPfF_Pmin_HMI					: REAL;				// JEMA P4 : AKUO P_Pmin

	ParamPfF_FhystLow_HMI				: REAL;				// JEMA fst1
	ParamPfF_FhystHigh_HMI				: REAL;				// JEMA fst2	
	
	
	ParamFreqRegSoCmax                  : REAL;
	ParamFreqRegSoCmin                  : REAL;
	                                    
	ParamTimeSoCRangeReachedRmp	       	: TIME;	 
	ParamTimeFreqRegStbDuration	       	: TIME;	 
	ParamTimeEnterStblPriorRmp	       	: TIME;  
                                       	 
                                       	 
	ParamTimeoutGridFormerTransition   	: TIME;	   
	ParamTimeoutGridFeederTransition	: TIME;  
    

	AX_BESS_Names						: ARRAY[1..CstNbESS_G] of string;                                    
	KK: INT;
	
	bConfirmPfF							: BOOL;
	bConfirmQfU							: BOOL;
END_VAR

FOR KK := 1 TO CstNbESS_G DO
	AX_BESS_Names[KK] := concat(STR1 := 'BESS', STR2 := INT_TO_STRING(KK));
END_FOR

//IF bResetParamQfU_PvF THEN
//	bResetParamQfU_PvF := FALSE;
//	
//	ParamPfF_FDbHigh_HMI 	:= A1_HPP.ParamPfF_FDbHigh;
//	ParamPfF_FDbLow_HMI 	:= A1_hpp.ParamPfF_FDbLow;
//	ParamPfF_FhystHigh_HMI 	:= A1_HPP.ParamPfF_FhystHigh;
//	ParamPfF_FhystLow_HMI 	:= A1_HPP.ParamPfF_FhystLow;
//	ParamPfF_Fmax_HMI		:= A1_HPP.ParamPfF_Fmax;
//	ParamPfF_Fmin_HMI		:= A1_HPP.ParamPfF_Fmin;
//	ParamPfF_PDbHigh_HMI 	:= A1_Hpp.ParamPfF_PDbHigh;
//	ParamPfF_PDbLow_HMI 	:= A1_hpp.ParamPfF_PDbLow;
//	ParamPfF_Pmax_HMI		:= A1_HPP.ParamPfF_Pmax;
//	ParamPfF_Pmin_HMI		:= A1_HPP.ParamPfF_Pmin;	
//	ParamQfU_QDbHigh_HMI	:= A1_HPP.ParamQfU_QDbHigh;
//	ParamQfU_QDbLow_HMI		:= A1_HPP.ParamQfU_QDbLow;
//	ParamQfU_Qmax_HMI		:= A1_HPP.ParamQfU_Qmax;
//	ParamQfU_Qmin_HMI		:= A1_HPP.ParamQfU_Qmin;
//	ParamQfU_UDbHigh_HMI	:= A1_HPP.ParamQfU_UDbHigh;
//	ParamQfU_UDbLow_HMI		:= A1_HPP.ParamQfU_UDbLow;
//	ParamQfU_Umax_HMI		:= A1_HPP.ParamQfU_Umax;
//	ParamQfU_Umin_HMI		:= A1_HPP.ParamQfU_Umin;	
//END_IF

// Param P(f)
	IF ParamPfF_FDbHigh_HMI >= ParamPfF_Fmax_HMI THEN
		ParamPfF_FDbHigh_HMI := ParamPfF_Fmax_HMI;
	END_IF
	paramPfF_PDbHigh_HMI 	:= 0;
	ParamPfF_PDbLow_HMI 	:= 0;
	
	IF ParamPfF_FDbLow_HMI <= ParamPfF_Fmin_HMI THEN
		ParamPfF_FDbLow_HMI := ParamPfF_Fmin_HMI;
	END_IF
		
	
	IF ParamPfF_FhystLow_HMI <= ParamPfF_FDbLow_HMI THEN
		ParamPfF_FhystLow_HMI := ParamPfF_FDbLow_HMI;
	END_IF 

	IF ParamPfF_FhystHigh_HMI >= ParamPfF_FDbHigh_HMI THEN
		ParamPfF_FhystHigh_HMI := ParamPfF_FDbHigh_HMI;
	END_IF 	
	
// Param Q(U)
	ParamQfU_QDbHigh_HMI 	:= 0;
	ParamQfU_QDbLow_HMI 	:= 0;
	
	IF ParamQfU_UDbHigh_HMI >= ParamQfU_Umax_HMI THEN
		ParamQfU_UDbHigh_HMI := ParamQfU_Umax_HMI;
	END_IF
	
	IF ParamQfU_UDbLow_HMI <= ParamQfU_Umin_HMI THEN
		ParamQfU_UDbLow_HMI := ParamQfU_Umin_HMI;
	END_IF
	
//IF bConfirmPfF THEN
//	bConfirmPfF := FALSE;	
//	A1_HPP.ParamPfF_PDbHigh		:= ParamPfF_PDbHigh_HMI;
//    A1_HPP.ParamPfF_Pmax		:= ParamPfF_Pmax_HMI;
//    A1_HPP.ParamPfF_PDbLow		:= ParamPfF_PDbLow_HMI;
//    A1_HPP.ParamPfF_Pmin		:= ParamPfF_Pmin_HMI;
//	
//	A1_HPP.ParamPfF_FDbHigh		:= ParamPfF_FDbHigh_HMI;
//    A1_HPP.ParamPfF_Fmax		:= ParamPfF_Fmax_HMI;
//    A1_HPP.ParamPfF_FDbLow		:= ParamPfF_FDbLow_HMI;
//    A1_HPP.ParamPfF_Fmin		:= ParamPfF_Fmin_HMI;
//	
//	A1_HPP.ParamPfF_FhystHigh	:= ParamPfF_FhystHigh_HMI;
//	A1_HPP.ParamPfF_FhystLow	:= ParamPfF_FhystLow_HMI;
//END_IF

//IF bConfirmQfU THEN	
//	bConfirmQfU := FALSE;
//	A1_HPP.ParamQfU_QDbHigh		:= ParamQfU_QDbHigh_HMI;
//    A1_HPP.ParamQfU_Qmax		:= ParamQfU_Qmax_HMI;
//    A1_HPP.ParamQfU_QDbLow		:= ParamQfU_QDbLow_HMI;
//    A1_HPP.ParamQfU_Qmin		:= ParamQfU_Qmin_HMI;
//	
//	A1_HPP.ParamQfU_UDbHigh		:= ParamQfU_UDbHigh_HMI;
//    A1_HPP.ParamQfU_Umax		:= ParamQfU_Umax_HMI;
//    A1_HPP.ParamQfU_UDbLow		:= ParamQfU_UDbLow_HMI;
//    A1_HPP.ParamQfU_Umin		:= ParamQfU_Umin_HMI;
//END_IF
//

IF PCS_RefreshValues THEN
	PCS_RefreshValues := FALSE;

	PCS1_ParamUnitID 						:= AX_ESS[bess_HMI.numEssDisplayed].AX_PCS[1].ParamUnitID 								;
	PCS1_ParamIPAddress			   			:= AX_ESS[bess_HMI.numEssDisplayed].AX_PCS[1].ParamIPAddress			   			    ;
	PCS1_ParamTcpPort						:= AX_ESS[bess_HMI.numEssDisplayed].AX_PCS[1].ParamTcpPort						        ;
	PCS1_ParamTempoComAlarm					:= AX_ESS[bess_HMI.numEssDisplayed].AX_PCS[1].ParamTempoComAlarm					    ;
	PCS1_ParamTempoComWarning				:= AX_ESS[bess_HMI.numEssDisplayed].AX_PCS[1].ParamTempoComWarning				        ;
	PCS1_ParamTimeOutBlckStrt          		:= AX_ESS[bess_HMI.numEssDisplayed].AX_PCS[1].ParamTimeOutBlckStrt          		    ;
	PCS1_ParamClockReadTime 				:= AX_ESS[bess_HMI.numEssDisplayed].AX_PCS[1].ParamClockReadTime 				        ;
	PCS1_ParamClockWriteTime 				:= AX_ESS[bess_HMI.numEssDisplayed].AX_PCS[1].ParamClockWriteTime 				        ;
	PCS1_ParamTimeout		            	:= AX_ESS[bess_HMI.numEssDisplayed].AX_PCS[1].ParamTimeout		            	        ;
	PCS1_ParamTimePulseTrig		    		:= AX_ESS[bess_HMI.numEssDisplayed].AX_PCS[1].ParamTimePulseTrig		    		    ;
	PCS1_ParamEssNum						:= AX_ESS[bess_HMI.numEssDisplayed].AX_PCS[1].ParamEssNum						        ;
	PCS1_ParamPcsNum						:= AX_ESS[bess_HMI.numEssDisplayed].AX_PCS[1].ParamPcsNum						        ;
	PCS1_ParamPoverQ						:= AX_ESS[bess_HMI.numEssDisplayed].AX_PCS[1].ParamPoverQ						        ;
	PCS1_ParamTimeSoCRangeReachedRmp		:= AX_ESS[bess_HMI.numEssDisplayed].AX_PCS[1].ParamTimeSoCRangeReachedRmp		        ;
	PCS1_ParamTimeFreqRegStbDuration		:= AX_ESS[bess_HMI.numEssDisplayed].AX_PCS[1].ParamTimeFreqRegStbDuration		        ;

	
	SBMS1_ParamClockWriteTime				:= AX_ESS[BESS_HMI.NumEssDisplayed].AX_BAT[1].ParamClockWriteTime;
	SBMS1_ParamIpAddress					:= AX_ESS[BESS_HMI.NumEssDisplayed].AX_BAT[1].ParamIpAddress;
	SBMS1_ParamTcpPort						:= AX_ESS[BESS_HMI.NumEssDisplayed].AX_BAT[1].ParamTcpPort;
	
	SBMS2_ParamClockWriteTime				:= AX_ESS[BESS_HMI.NumEssDisplayed].AX_BAT[2].ParamClockWriteTime;
	SBMS2_ParamIpAddress					:= AX_ESS[BESS_HMI.NumEssDisplayed].AX_BAT[2].ParamIpAddress;
	SBMS2_ParamTcpPort						:= AX_ESS[BESS_HMI.NumEssDisplayed].AX_BAT[2].ParamTcpPort;
	
END_IF


IF PCS1_bParamUnitID 						THEN AX_ESS[Bess_hmi.NumEssDisplayed].AX_PCS[1].ParamUnitID := PCS1_ParamUnitID; PCS1_bParamUnitID := FALSE; END_IF 
IF PCS1_bParamIPAddress 					THEN AX_ESS[Bess_hmi.NumEssDisplayed].AX_PCS[1].ParamIPAddress := PCS1_ParamIPAddress; PCS1_bParamIPAddress := FALSE; END_IF 
IF PCS1_bParamTcpPort 						THEN AX_ESS[Bess_hmi.NumEssDisplayed].AX_PCS[1].ParamTcpPort := PCS1_ParamTcpPort; PCS1_bParamTcpPort := FALSE; END_IF 
IF PCS1_bParamTempoComAlarm 				THEN AX_ESS[Bess_hmi.NumEssDisplayed].AX_PCS[1].ParamTempoComAlarm := PCS1_ParamTempoComAlarm; PCS1_bParamTempoComAlarm := FALSE; END_IF 
IF PCS1_bParamTempoComWarning 				THEN AX_ESS[Bess_hmi.NumEssDisplayed].AX_PCS[1].ParamTempoComWarning := PCS1_ParamTempoComWarning; PCS1_bParamTempoComWarning := FALSE; END_IF 
IF PCS1_bParamTimeOutBlckStrt   			THEN AX_ESS[Bess_hmi.NumEssDisplayed].AX_PCS[1].ParamTimeOutBlckStrt           := PCS1_ParamTimeOutBlckStrt          ; PCS1_bParamTimeOutBlckStrt           := FALSE; END_IF 
IF PCS1_bParamClockReadTime  				THEN AX_ESS[Bess_hmi.NumEssDisplayed].AX_PCS[1].ParamClockReadTime  := PCS1_ParamClockReadTime ; PCS1_bParamClockReadTime  := FALSE; END_IF 
IF PCS1_bParamClockWriteTime  				THEN AX_ESS[Bess_hmi.NumEssDisplayed].AX_PCS[1].ParamClockWriteTime  := PCS1_ParamClockWriteTime ; PCS1_bParamClockWriteTime  := FALSE; END_IF 
IF PCS1_bParamTimeout 						THEN AX_ESS[Bess_hmi.NumEssDisplayed].AX_PCS[1].ParamTimeout := PCS1_ParamTimeout; PCS1_bParamTimeout := FALSE; END_IF 
IF PCS1_bParamEssNum 						THEN AX_ESS[Bess_hmi.NumEssDisplayed].AX_PCS[1].ParamEssNum := PCS1_ParamEssNum; PCS1_bParamEssNum := FALSE; END_IF 
IF PCS1_bParamPcsNum 						THEN AX_ESS[Bess_hmi.NumEssDisplayed].AX_PCS[1].ParamPcsNum := PCS1_ParamPcsNum; PCS1_bParamPcsNum := FALSE; END_IF 
IF PCS1_bParamPoverQ 						THEN AX_ESS[Bess_hmi.NumEssDisplayed].AX_PCS[1].ParamPoverQ := PCS1_ParamPoverQ; PCS1_bParamPoverQ := FALSE; END_IF 
IF PCS1_bParamTimeSoCRangeReachedRmp 		THEN AX_ESS[Bess_hmi.NumEssDisplayed].AX_PCS[1].ParamTimeSoCRangeReachedRmp := PCS1_ParamTimeSoCRangeReachedRmp; PCS1_bParamTimeSoCRangeReachedRmp := FALSE; END_IF 
IF PCS1_bParamTimeFreqRegStbDuration 		THEN AX_ESS[Bess_hmi.NumEssDisplayed].AX_PCS[1].ParamTimeFreqRegStbDuration := PCS1_ParamTimeFreqRegStbDuration; PCS1_bParamTimeFreqRegStbDuration := FALSE; END_IF

END_PROGRAM

// ---- 04_Application/HMI/Parameters/ParamEMS.TcPOU
PROGRAM ParamEMS
VAR CONSTANT
	MaxNumberBess 	: UINT := 5;
	MaxNumberGen 	: UINT := 20;
	MaxNumberLoad 	: UINT := 1;
	MaxNumberRen	: UINT := 20;
END_VAR

VAR
	
	bChangeBess				: BOOL;
	bChangeGen				: BOOL;
	bChangeLoad				: BOOL;
	bChangeRen				: BOOL;
	
	TRIG_ChangeBess			: R_TRIG;
	TRIG_ChangeGen			: R_TRIG;
	TRIG_ChangeLoad			: R_TRIG;
	TRIG_ChangeRen			: R_TRIG;
	
	NumBessDisplayed 		: UINT:= 1;
	NumGenDisplayed 		: UINT:= 1;
	NumLoadDisplayed 		: UINT:= 1;
	NumRenDisplayed 		: UINT:= 1;
	
	NumBessDisplayed_Old	: UINT:= 1;
	NumGenDisplayed_Old		: UINT:= 1;
	NumLoadDisplayed_Old	: UINT:= 1;
	NumRenDisplayed_Old		: UINT:= 1;
	
	NameBessDisplayed		: STRING;
	NameGenDisplayed		: STRING;
	NameLoadDisplayed		: STRING;
	NameRenDisplayed		: STRING;
	
	BessNames 				: ARRAY[1.. MaxNumberBess] OF STRING;
	GenNames 				: ARRAY[1..MaxNumberGen] OF STRING;
	LoadNames 				: ARRAY[1..MaxNumberLoad] OF STRING;
	RenNames				: ARRAY[1..MaxNumberRen] OF STRING;
	
	// INPUTS 
		// LOAD
			Load_IN_P	 			: REAL;
			Load_IN_Q				: REAL;
		// BESS
			Bess_IN_MesS			: REAL;
			Bess_IN_MesP			: REAL;
			Bess_IN_MesQ			: REAL;
			Bess_IN_MesSoC			: REAL;
			Bess_IN_MesPmax			: REAL;
			Bess_IN_MesPmin			: REAL;
			Bess_IN_MesQmax			: REAL;
			Bess_IN_MesQmin			: REAL;
		// GEN
			Gen_IN_Mode				: WORD;
			Gen_IN_Prio				: UINT;
			Gen_IN_RunHour			: REAL;
			Gen_IN_P				: REAL;
			Gen_IN_Q				: REAL;
		// REN	
			Ren_IN_MesP				: REAL;
			Ren_IN_MesQ				: REAL;
			Ren_IN_Prio				: UINT;

	// OUTPUTS 	
		// BESS
			Bess_OUT_SetptP			: REAL;
			Bess_OUT_SetptQ			: REAL;
		// GEN	
			Gen_OUT_setptP			: REAL;
			Gen_OUT_setptQ			: REAL;
		// REN
			Ren_Out_SetptP			: REAL;
	
	KK: UINT;
END_VAR

TRIG_ChangeBess(CLK := bChangeBess);
TRIG_ChangeGen(CLK := bChangeGen);
TRIG_ChangeLoad(CLK := bChangeLoad);
TRIG_ChangeRen(CLK := bChangeRen);

END_PROGRAM

// ---- 04_Application/MAIN/POU.TcPOU
FUNCTION_BLOCK POU
VAR_INPUT
END_VAR
VAR_OUTPUT
END_VAR
VAR

END_VAR

END_FUNCTION_BLOCK
